{attribute 'GeneratedUsingTerminal: EL4712--0000'}
{attribute addProperty BoxType "EL4712--0000"}
{attribute addProperty Id "Ch2_CycleCountAT %Q*UINT2"}
{attribute addProperty CRC "35773855"}
{attribute addProperty Size "2"}
TYPE Ch2_CycleCount_0221DD9F :
STRUCT
	{attribute addProperty Name "Ch2_CycleCount"}
	Ch2_CycleCount AT %Q* : UINT;
END_STRUCT
END_TYPE

(* stored: Version 1.2.0.0, ProductVersion 3.1.4024.9
   DUT Ch2_CycleCount_0221DD9F: Id {01246e2a-49c4-4b5e-a7a7-728c2d2ebc0c} *)
